{attribute 'linkalways'} 
{attribute 'no_explicit_call' := 'This FB is a CLASS and must be accessed using methods or properties'}
{attribute 'enable_dynamic_creation'}
FUNCTION_BLOCK ABSTRACT QueueEvent EXTENDS Disposable
VAR
	_targetQueue : I_Queue;
END_VAR

METHOD FB_init : BOOL
VAR_INPUT
	bInitRetains : BOOL; // if TRUE, the retain variables are initialized (warm start / cold start)
	bInCopyCode : BOOL;  // if TRUE, the instance afterwards gets moved into the copy code (online change)
	TargetQueue : I_Queue;
END_VAR
THIS^._targetQueue := TargetQueue;
END_METHOD

PROPERTY PUBLIC TargetQueue : I_Queue
GET // PUBLIC
TargetQueue := _targetQueue;
END_GET
END_PROPERTY

END_FUNCTION_BLOCK

(* stored: Version 1.1.0.1, ProductVersion 3.1.4024.12
   POU QueueEvent: Id {a68f9214-e069-4039-ab91-9e781278d499}, SpecialFunc None
   Folder Constructor: Id {1e676b3b-ec17-43d8-84e0-efb28fa66654}
   Method FB_init: Id {e7c4e2ea-89c1-438b-883d-ad31615df81b}
   Property TargetQueue: Id {d1356c9e-dbd3-4c0b-8017-b4b4878374ca}
   Get Get: Id {7dcd490e-d578-4f49-81d3-9bcfcf887cc5} *)
